{attribute 'pack_mode' := '1'}
TYPE TPositionXYTheta :
STRUCT
	lrX		: LREAL;
	lrY		: LREAL;
	lrTheta	: LREAL;
END_STRUCT
END_TYPE

(* stored: Version 1.1.0.1, ProductVersion 3.1.4022.12
   DUT TPositionXYTheta: Id {82e4e827-5cc5-44f5-9fe5-48de8bd564c2} *)
